// TIA Portal project "S7-1500 Otopark" (V18)

(* hardware
DEVICE "S7-1500/ET200MP station_1"  S7-1500 station
   slot 0: "Rail_0"  Rack  6ES7 590-1***0-0AA0
   slot 1: "PLC_1"  CPU 1512C-1 PN  6ES7 512-1CK01-0AB0  V2.8
      slot 3: "CPU display_1"  6ES7591-1AA00-0AA0
      slot 32768: "PROFINET interface_1"  X1
         slot 32769: "Port_1"  X1 P1
         slot 32770: "Port_2"  X1 P2
      slot 34817: "Virtual CP interface port_1"  Virtual CP interface port  Virtual CP interface port
DEVICE "HMI_1"  KTP700 Basic PN
   slot 0: "HMI_1"  KTP700 Basic PN  6AV2 123-2GB03-0AX0  14.0.1.0
   slot 1: "HMI_RT_1"  KTP700 Basic PN  6AV2 123-2GB03-0AX0  14.0.1.0
   slot 5: "HMI_1.IE_CP_1"  PROFINET Interface  14.0.1.0
      slot 1: "PROFINET Interface_1"  PROFINET Interface
         slot 1: "Port_1"  Port
*)

// ===== PLC "PLC_1"  CPU 1512C-1 PN =====

VAR_GLOBAL   // PLC tag table "Default tag table"
   "Otopark Dolu" AT %Q0.0 : Bool;
   "Reset" AT %I0.0 : Bool;
   "Arttır" AT %I0.1 : Bool;
   "Azalt" AT %I0.2 : Bool;
   "Uyarı" AT %M0.0 : Bool;
   "Araç Sayısı" AT %MW2 : Int;
   "Otopark Boş" AT %Q0.1 : Bool;
   "boş" AT %MW4 : Int;
END_VAR

// folder: System blocks/Program resources

DATA_BLOCK "IEC_Counter_0_DB"   // DB1
{ S7_Optimized_Access := 'TRUE' }
AUTHOR : Simatic
FAMILY : IEC
NAME : CNTR
VERSION : 1.0
// stored: InstanceOfName IEC_COUNTER
"IEC_COUNTER"
BEGIN
END_DATA_BLOCK

// folder: (top level)

ORGANIZATION_BLOCK "Main"   // OB1, LAD, ProgramCycle
TITLE = "Main Program Sweep (Cycle)"
{ S7_Optimized_Access := 'TRUE' }
VERSION : 0.1
   VAR_INPUT
      Initial_Call : Bool;   // Initial call of this OB
      Remanence : Bool;   // =True, if remanent data are available
   END_VAR
BEGIN

REGION Network 1
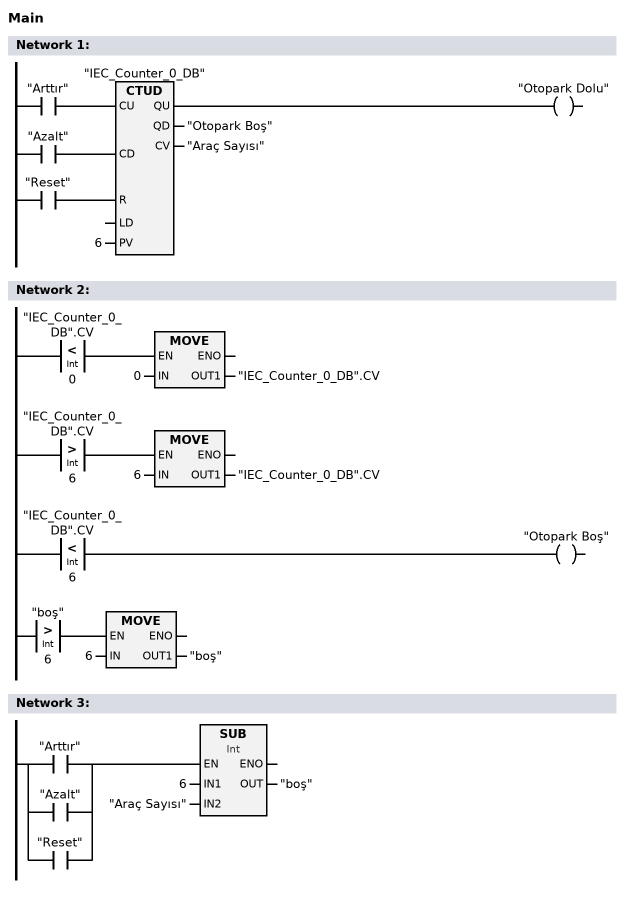
   "IEC_Counter_0_DB".CTUD(CU := "Arttır",
                           CD := "Azalt",
                           R := "Reset",
                           PV := 6,
                           QD => "Otopark Boş",
                           CV => "Araç Sayısı");
   "Otopark Dolu" := "IEC_Counter_0_DB".QU;
END_REGION

REGION Network 2
   RUNG wire#powerrail
      { S7_Templates := "SrcType := Int" } LT_Contact(in1 := "IEC_Counter_0_DB".CV, in2 := 0)
      Move(in := 0, out1 => "IEC_Counter_0_DB".CV)
   END_RUNG
   RUNG wire#powerrail
      { S7_Templates := "SrcType := Int" } GT_Contact(in1 := "IEC_Counter_0_DB".CV, in2 := 6)
      Move(in := 6, out1 => "IEC_Counter_0_DB".CV)
   END_RUNG
   RUNG wire#powerrail
      { S7_Templates := "SrcType := Int" } LT_Contact(in1 := "IEC_Counter_0_DB".CV, in2 := 6)
      Coil( "Otopark Boş" )
   END_RUNG
   RUNG wire#powerrail
      { S7_Templates := "SrcType := Int" } GT_Contact(in1 := "boş", in2 := 6)
      Move(in := 6, out1 => "boş")
   END_RUNG
   // the same network as SCL:
   IF "IEC_Counter_0_DB".CV < 0 THEN "IEC_Counter_0_DB".CV := 0; END_IF;
   IF "IEC_Counter_0_DB".CV > 6 THEN "IEC_Counter_0_DB".CV := 6; END_IF;
   "Otopark Boş" := "IEC_Counter_0_DB".CV < 6;
   IF "boş" > 6 THEN "boş" := 6; END_IF;
END_REGION

REGION Network 3
   RUNG wire#powerrail
      Contact( "Arttır" )
      wire#w1
      { S7_Templates := "SrcType := Int" } Sub(in1 := 6, in2 := "Araç Sayısı", out => "boş")
   END_RUNG
   RUNG wire#powerrail
      Contact( "Azalt" )
   END_RUNG wire#w1
   RUNG wire#powerrail
      Contact( "Reset" )
   END_RUNG wire#w1
   // the same network as SCL:
   IF "Arttır" OR "Azalt" OR "Reset" THEN "boş" := 6 - "Araç Sayısı"; END_IF;
END_REGION
END_ORGANIZATION_BLOCK

(* ===== HMI "HMI_RT_1" =====
system functions are stored by id; their names below are inferred from use
connection "Connection_1": ETHERNET, SMART_S7_1500_OMS
connection "HMI_Connection_1": ETHERNET, SMART_S7_1500_OMS

HMI tags "Default tag table"
   "Tag_ScreenNumber" : UInt, internal
   "Arttır" : Bool = PLC Arttır AT %I0.1, 100 ms
   "Azalt" : Bool = PLC Azalt AT %I0.2, 100 ms
   "Reset" : Bool = PLC Reset AT %I0.0, 100 ms
   "Araç Sayısı" : Int = PLC "Araç Sayısı" AT %MW2, 100 ms
   "Otopark Dolu" : Bool = PLC "Otopark Dolu" AT %Q0.0, 100 ms
   "boş" : Int = PLC boş AT %MW4, 100 ms

graphic list "OtoparkDolu": 1 'Graphic_5'; 0 'Graphic_4'

Template "Template_1" 800x480
   Button "Exit" at 714,429 size 71x50; TextOff 'Exit'; PictureOff "ExitRuntime_KTP700_Basic_PN_TR"; PictureOn "ExitRuntime_KTP700_Basic_PN_TR"
      on Release: StopRuntime(0)
   Button "Language" at 614,429 size 71x50; TextOff 'Language'; PictureOff "ToggleLanguage_KTP700_Basic_PN_TR"; PictureOn "ToggleLanguage_KTP700_Basic_PN_TR"
      on Release: function_fb9197e8(-1)
   Button "Log on" at 514,429 size 71x50; TextOff 'Log on'; PictureOff "Login_KTP700_Basic_PN_TR"; PictureOn "Login_KTP700_Basic_PN_TR"
      on Release: function_a2a04561()
   Button "Alarms" at 114,429 size 71x50; TextOff 'Alarms'; PictureOff "AlarmDisplay_KTP700_Basic_PN_TR"; PictureOn "AlarmDisplay_KTP700_Basic_PN_TR"
      on Release: function_ef3f5d25("Alarm window_Unacknowledged", -1)
   Button "Start screen" at 14,429 size 71x50; TextOff 'Start screen'; PictureOff "NavigateHome_KTP700_Basic_PN_TR"; PictureOn "NavigateHome_KTP700_Basic_PN_TR"
      on Release: ActivateScreen("Root screen", 0)
   SymbolicIOField "Symbolic_IO_Field_Screen" at 93,9 size 600x33; TextOff '0'; TextOn '1'; TextList "TextList_ScreenNames"
      ProcessValue <- "Tag_ScreenNumber"
      on Change: ActivateScreenByNumber("Tag_ScreenNumber", 0)
   DateTimeField "HmiScreenItemData" at 695,25 size 105x25
   DateTimeField "HmiScreenItemData_1" at 695,0 size 105x25
   GraphicView "Logo" at 0,0 size 91x51; Picture "Logo of HMI_1"

screen "Root screen" 800x480, template "Template_1"
   on GenerateScreen: SetTag("Tag_ScreenNumber", 1)
   TextField "HmiScreenItemData" at 0,63 size 644x25; Text 'S7-1500 PLC Eğitim Seti Otopark Projesi'
   Button "Button_1" at 92,130 size 141x79; TextOff 'Arttır'
      on Press: SetBit("Arttır")
      on Release: ResetBit("Arttır")
   Button "Button_2" at 92,325 size 141x79; TextOff 'Reset'
      on Press: SetBit("Reset")
      on Release: ResetBit("Reset")
   Button "Button_3" at 92,227 size 141x79; TextOff 'Azalt'
      on Press: SetBit("Azalt")
      on Release: ResetBit("Azalt")
   IOField "I/O field_1" at 493,333 size 96x32; FormatPattern s99999
      ProcessValue <- "Araç Sayısı"
   GraphicIOField "Graphic I/O field_1" at 283,148 size 306x185; PictureList "OtoparkDolu"
      ProcessValue <- "Otopark Dolu"
   IOField "I/O field_2" at 493,372 size 96x32; FormatPattern s99999
      ProcessValue <- "boş"
   TextField "Text field_1" at 285,333 size 171x32; Text 'Araç Sayısı-->'
   TextField "Text field_2" at 279,372 size 207x32; Text 'Boş Yer Sayısı-->'
   TextField "Text field_3" at 341,125 size 199x23; Text 'Park Etmeye Uygunluk?'
*)